Staubli VAL3: onRun.pgx

public program onRun(string& x_sItem[])
  local num l_nResult
begin
  //
  call loadIt("_"+x_sItem)
  //
end
